// TIA Portal V17 export
// export: Created 2025-03-07T09:17:10.7987229Z, ExportSetting WithDefaults, DisplayName Totally Integrated Automation Portal, DisplayVersion V17 Update 8, DisplayName TIA Portal Openness, DisplayVersion V17 Update 8, DisplayName TIA Portal Version Control Interface, DisplayVersion V17, DisplayName SINAMICS Startdrive Advanced, DisplayVersion V17 SP2, DisplayName SINAMICS Startdrive G110M, G120, G120C, G120D, G120P, G115D, DisplayVersion V17 SP2, DisplayName SINAMICS Startdrive G130, G150, S120, S150, SINAMICS MV, S210, DisplayVersion V17 SP2, DisplayName STEP 7 Professional, DisplayVersion V17 Update 8, DisplayName SINUMERIK ONE STEP 7 Toolbox, DisplayVersion V17 Update 12, DisplayName SINUMERIK 840D sl STEP 7 Toolbox, DisplayVersion V17 Update 12, DisplayName STEP 7 Safety, DisplayVersion V17 Update 6, DisplayName WinCC Advanced, DisplayVersion V17 Update 8
FUNCTION "FC321_CHANNEL_1" : Void   // FC321, LAD
{ S7_Optimized_Access := 'FALSE' }
AUTHOR : ETXETAR
VERSION : 1.0
// stored: AutoNumber false, IsIECCheckEnabled false, SetENOAutomatically false, UDAEnableTagReadback false
BEGIN

REGION Network 1: RESET CHANNEL 1 / CHANNEL 1 (NC RESET - NC START)
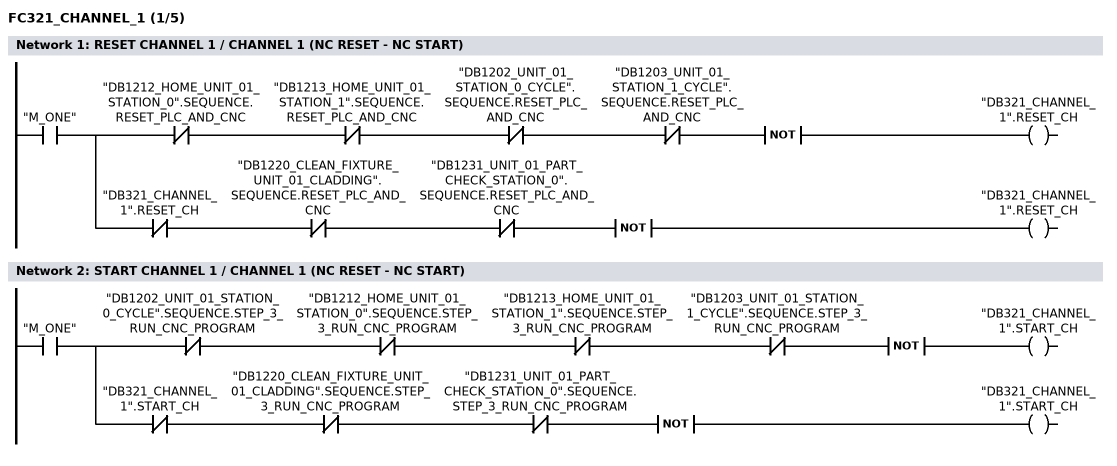
   RUNG wire#powerrail
      Contact( "M_ONE" )
      wire#w1
      I_Contact( "DB1212_HOME_UNIT_01_STATION_0".SEQUENCE.RESET_PLC_AND_CNC )
      I_Contact( "DB1213_HOME_UNIT_01_STATION_1".SEQUENCE.RESET_PLC_AND_CNC )
      I_Contact( "DB1202_UNIT_01_STATION_0_CYCLE".SEQUENCE.RESET_PLC_AND_CNC )
      I_Contact( "DB1203_UNIT_01_STATION_1_CYCLE".SEQUENCE.RESET_PLC_AND_CNC )
      Not()
      Coil( "DB321_CHANNEL_1".RESET_CH )
   END_RUNG
   RUNG wire#w1
      I_Contact( "DB321_CHANNEL_1".RESET_CH )
      I_Contact( "DB1220_CLEAN_FIXTURE_UNIT_01_CLADDING".SEQUENCE.RESET_PLC_AND_CNC )
      I_Contact( "DB1231_UNIT_01_PART_CHECK_STATION_0".SEQUENCE.RESET_PLC_AND_CNC )
      Not()
      Coil( "DB321_CHANNEL_1".RESET_CH )
   END_RUNG
   // the same network as SCL:
   "DB321_CHANNEL_1".RESET_CH := NOT ("M_ONE" AND NOT "DB1212_HOME_UNIT_01_STATION_0".SEQUENCE.RESET_PLC_AND_CNC AND NOT "DB1213_HOME_UNIT_01_STATION_1".SEQUENCE.RESET_PLC_AND_CNC AND NOT "DB1202_UNIT_01_STATION_0_CYCLE".SEQUENCE.RESET_PLC_AND_CNC AND NOT "DB1203_UNIT_01_STATION_1_CYCLE".SEQUENCE.RESET_PLC_AND_CNC);
   "DB321_CHANNEL_1".RESET_CH := NOT ("M_ONE" AND NOT "DB321_CHANNEL_1".RESET_CH AND NOT "DB1220_CLEAN_FIXTURE_UNIT_01_CLADDING".SEQUENCE.RESET_PLC_AND_CNC AND NOT "DB1231_UNIT_01_PART_CHECK_STATION_0".SEQUENCE.RESET_PLC_AND_CNC);
END_REGION

REGION Network 2: START CHANNEL 1 / CHANNEL 1 (NC RESET - NC START)
   RUNG wire#powerrail
      Contact( "M_ONE" )
      wire#w1
      I_Contact( "DB1202_UNIT_01_STATION_0_CYCLE".SEQUENCE.STEP_3_RUN_CNC_PROGRAM )
      I_Contact( "DB1212_HOME_UNIT_01_STATION_0".SEQUENCE.STEP_3_RUN_CNC_PROGRAM )
      I_Contact( "DB1213_HOME_UNIT_01_STATION_1".SEQUENCE.STEP_3_RUN_CNC_PROGRAM )
      I_Contact( "DB1203_UNIT_01_STATION_1_CYCLE".SEQUENCE.STEP_3_RUN_CNC_PROGRAM )
      Not()
      Coil( "DB321_CHANNEL_1".START_CH )
   END_RUNG
   RUNG wire#w1
      I_Contact( "DB321_CHANNEL_1".START_CH )
      I_Contact( "DB1220_CLEAN_FIXTURE_UNIT_01_CLADDING".SEQUENCE.STEP_3_RUN_CNC_PROGRAM )
      I_Contact( "DB1231_UNIT_01_PART_CHECK_STATION_0".SEQUENCE.STEP_3_RUN_CNC_PROGRAM )
      Not()
      Coil( "DB321_CHANNEL_1".START_CH )
   END_RUNG
   // the same network as SCL:
   "DB321_CHANNEL_1".START_CH := NOT ("M_ONE" AND NOT "DB1202_UNIT_01_STATION_0_CYCLE".SEQUENCE.STEP_3_RUN_CNC_PROGRAM AND NOT "DB1212_HOME_UNIT_01_STATION_0".SEQUENCE.STEP_3_RUN_CNC_PROGRAM AND NOT "DB1213_HOME_UNIT_01_STATION_1".SEQUENCE.STEP_3_RUN_CNC_PROGRAM AND NOT "DB1203_UNIT_01_STATION_1_CYCLE".SEQUENCE.STEP_3_RUN_CNC_PROGRAM);
   "DB321_CHANNEL_1".START_CH := NOT ("M_ONE" AND NOT "DB321_CHANNEL_1".START_CH AND NOT "DB1220_CLEAN_FIXTURE_UNIT_01_CLADDING".SEQUENCE.STEP_3_RUN_CNC_PROGRAM AND NOT "DB1231_UNIT_01_PART_CHECK_STATION_0".SEQUENCE.STEP_3_RUN_CNC_PROGRAM);
END_REGION

REGION Network 3: CALL FB321 CHANNEL 1
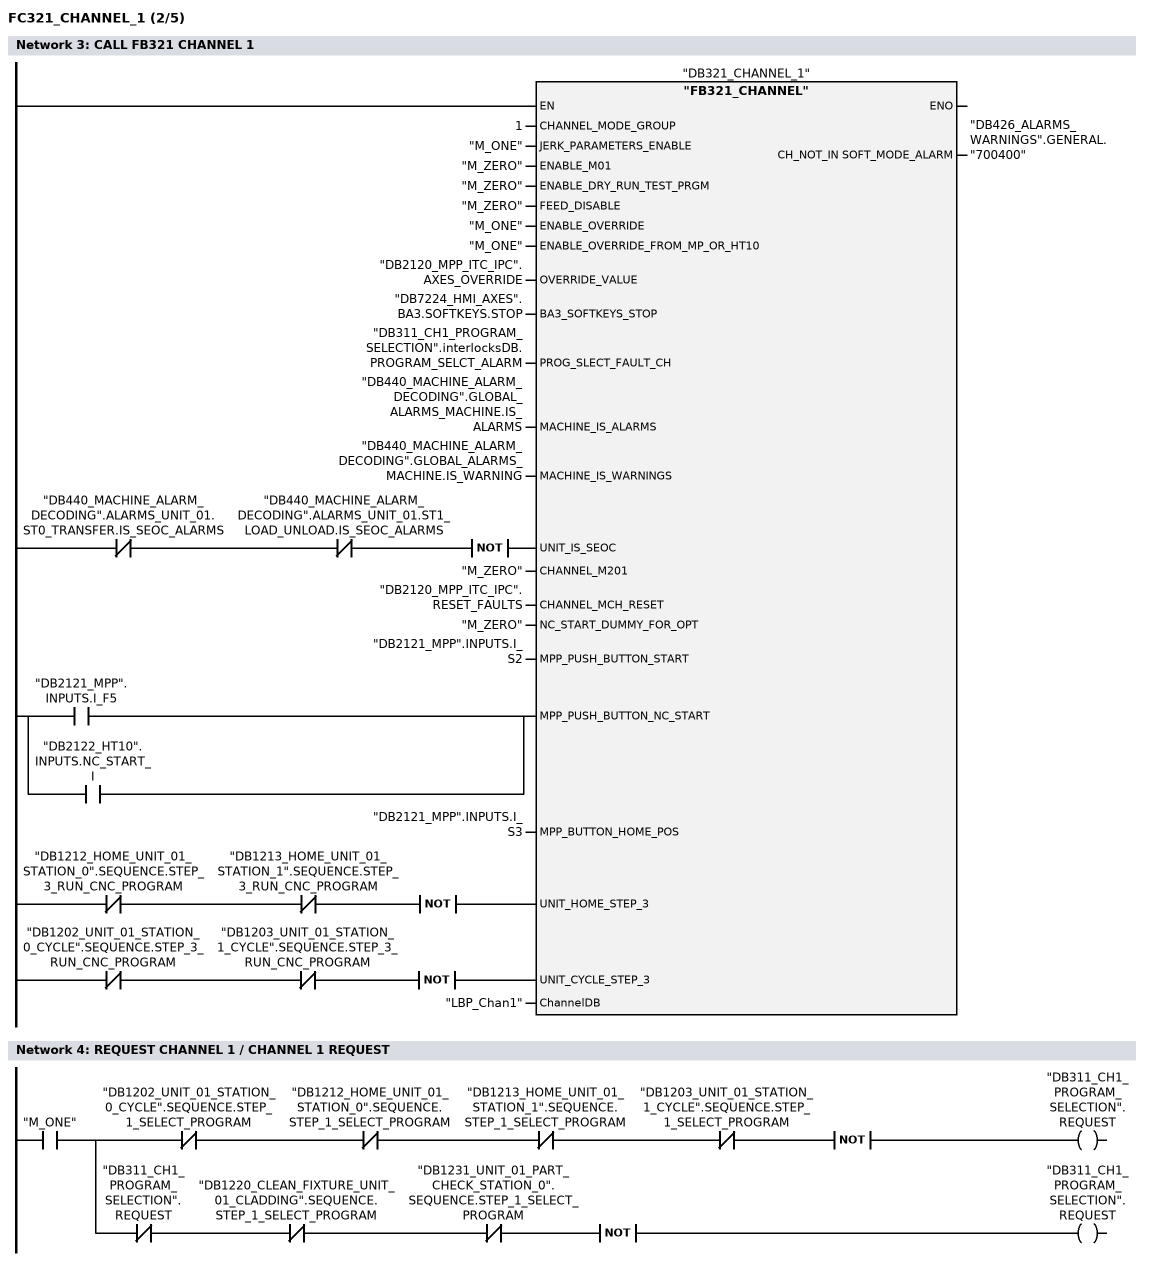
   RUNG wire#powerrail
      "DB321_CHANNEL_1"(UNIT_IS_SEOC := wire#w1, MPP_PUSH_BUTTON_NC_START := wire#w2, UNIT_HOME_STEP_3 := wire#w3, UNIT_CYCLE_STEP_3 := wire#w4, CHANNEL_MODE_GROUP := 1, JERK_PARAMETERS_ENABLE := "M_ONE", ENABLE_M01 := "M_ZERO", ENABLE_DRY_RUN_TEST_PRGM := "M_ZERO", FEED_DISABLE := "M_ZERO", ENABLE_OVERRIDE := "M_ONE", ENABLE_OVERRIDE_FROM_MP_OR_HT10 := "M_ONE", OVERRIDE_VALUE := "DB2120_MPP_ITC_IPC".AXES_OVERRIDE, BA3_SOFTKEYS_STOP := "DB7224_HMI_AXES".BA3.SOFTKEYS.STOP, PROG_SLECT_FAULT_CH := "DB311_CH1_PROGRAM_SELECTION".interlocksDB.PROGRAM_SELCT_ALARM, MACHINE_IS_ALARMS := "DB440_MACHINE_ALARM_DECODING".GLOBAL_ALARMS_MACHINE.IS_ALARMS, MACHINE_IS_WARNINGS := "DB440_MACHINE_ALARM_DECODING".GLOBAL_ALARMS_MACHINE.IS_WARNING, CHANNEL_M201 := "M_ZERO", CHANNEL_MCH_RESET := "DB2120_MPP_ITC_IPC".RESET_FAULTS, NC_START_DUMMY_FOR_OPT := "M_ZERO", MPP_PUSH_BUTTON_START := "DB2121_MPP".INPUTS.I_S2, MPP_BUTTON_HOME_POS := "DB2121_MPP".INPUTS.I_S3, ChannelDB := "LBP_Chan1", "CH_NOT_IN SOFT_MODE_ALARM" => "DB426_ALARMS_WARNINGS".GENERAL."700400")
   END_RUNG
   RUNG wire#powerrail
      I_Contact( "DB440_MACHINE_ALARM_DECODING".ALARMS_UNIT_01.ST0_TRANSFER.IS_SEOC_ALARMS )
      I_Contact( "DB440_MACHINE_ALARM_DECODING".ALARMS_UNIT_01.ST1_LOAD_UNLOAD.IS_SEOC_ALARMS )
      Not()
   END_RUNG wire#w1
   RUNG wire#powerrail
      Contact( "DB2121_MPP".INPUTS.I_F5 )
   END_RUNG wire#w2
   RUNG wire#powerrail
      Contact( "DB2122_HT10".INPUTS.NC_START_I )
   END_RUNG wire#w2
   RUNG wire#powerrail
      I_Contact( "DB1212_HOME_UNIT_01_STATION_0".SEQUENCE.STEP_3_RUN_CNC_PROGRAM )
      I_Contact( "DB1213_HOME_UNIT_01_STATION_1".SEQUENCE.STEP_3_RUN_CNC_PROGRAM )
      Not()
   END_RUNG wire#w3
   RUNG wire#powerrail
      I_Contact( "DB1202_UNIT_01_STATION_0_CYCLE".SEQUENCE.STEP_3_RUN_CNC_PROGRAM )
      I_Contact( "DB1203_UNIT_01_STATION_1_CYCLE".SEQUENCE.STEP_3_RUN_CNC_PROGRAM )
      Not()
   END_RUNG wire#w4
   // the same network as SCL:
   "DB321_CHANNEL_1"(CHANNEL_MODE_GROUP := 1,   // "FB321_CHANNEL"
                     JERK_PARAMETERS_ENABLE := "M_ONE",
                     ENABLE_M01 := "M_ZERO",
                     ENABLE_DRY_RUN_TEST_PRGM := "M_ZERO",
                     FEED_DISABLE := "M_ZERO",
                     ENABLE_OVERRIDE := "M_ONE",
                     ENABLE_OVERRIDE_FROM_MP_OR_HT10 := "M_ONE",
                     OVERRIDE_VALUE := "DB2120_MPP_ITC_IPC".AXES_OVERRIDE,
                     BA3_SOFTKEYS_STOP := "DB7224_HMI_AXES".BA3.SOFTKEYS.STOP,
                     PROG_SLECT_FAULT_CH := "DB311_CH1_PROGRAM_SELECTION".interlocksDB.PROGRAM_SELCT_ALARM,
                     MACHINE_IS_ALARMS := "DB440_MACHINE_ALARM_DECODING".GLOBAL_ALARMS_MACHINE.IS_ALARMS,
                     MACHINE_IS_WARNINGS := "DB440_MACHINE_ALARM_DECODING".GLOBAL_ALARMS_MACHINE.IS_WARNING,
                     UNIT_IS_SEOC := NOT (NOT "DB440_MACHINE_ALARM_DECODING".ALARMS_UNIT_01.ST0_TRANSFER.IS_SEOC_ALARMS AND NOT "DB440_MACHINE_ALARM_DECODING".ALARMS_UNIT_01.ST1_LOAD_UNLOAD.IS_SEOC_ALARMS),
                     CHANNEL_M201 := "M_ZERO",
                     CHANNEL_MCH_RESET := "DB2120_MPP_ITC_IPC".RESET_FAULTS,
                     NC_START_DUMMY_FOR_OPT := "M_ZERO",
                     MPP_PUSH_BUTTON_START := "DB2121_MPP".INPUTS.I_S2,
                     MPP_PUSH_BUTTON_NC_START := "DB2121_MPP".INPUTS.I_F5 OR "DB2122_HT10".INPUTS.NC_START_I,
                     MPP_BUTTON_HOME_POS := "DB2121_MPP".INPUTS.I_S3,
                     UNIT_HOME_STEP_3 := NOT (NOT "DB1212_HOME_UNIT_01_STATION_0".SEQUENCE.STEP_3_RUN_CNC_PROGRAM AND NOT "DB1213_HOME_UNIT_01_STATION_1".SEQUENCE.STEP_3_RUN_CNC_PROGRAM),
                     UNIT_CYCLE_STEP_3 := NOT (NOT "DB1202_UNIT_01_STATION_0_CYCLE".SEQUENCE.STEP_3_RUN_CNC_PROGRAM AND NOT "DB1203_UNIT_01_STATION_1_CYCLE".SEQUENCE.STEP_3_RUN_CNC_PROGRAM),
                     ChannelDB := "LBP_Chan1",
                     "CH_NOT_IN SOFT_MODE_ALARM" => "DB426_ALARMS_WARNINGS".GENERAL."700400");
END_REGION

REGION Network 4: REQUEST CHANNEL 1 / CHANNEL 1 REQUEST
   RUNG wire#powerrail
      Contact( "M_ONE" )
      wire#w1
      I_Contact( "DB1202_UNIT_01_STATION_0_CYCLE".SEQUENCE.STEP_1_SELECT_PROGRAM )
      I_Contact( "DB1212_HOME_UNIT_01_STATION_0".SEQUENCE.STEP_1_SELECT_PROGRAM )
      I_Contact( "DB1213_HOME_UNIT_01_STATION_1".SEQUENCE.STEP_1_SELECT_PROGRAM )
      I_Contact( "DB1203_UNIT_01_STATION_1_CYCLE".SEQUENCE.STEP_1_SELECT_PROGRAM )
      Not()
      Coil( "DB311_CH1_PROGRAM_SELECTION".REQUEST )
   END_RUNG
   RUNG wire#w1
      I_Contact( "DB311_CH1_PROGRAM_SELECTION".REQUEST )
      I_Contact( "DB1220_CLEAN_FIXTURE_UNIT_01_CLADDING".SEQUENCE.STEP_1_SELECT_PROGRAM )
      I_Contact( "DB1231_UNIT_01_PART_CHECK_STATION_0".SEQUENCE.STEP_1_SELECT_PROGRAM )
      Not()
      Coil( "DB311_CH1_PROGRAM_SELECTION".REQUEST )
   END_RUNG
   // the same network as SCL:
   "DB311_CH1_PROGRAM_SELECTION".REQUEST := NOT ("M_ONE" AND NOT "DB1202_UNIT_01_STATION_0_CYCLE".SEQUENCE.STEP_1_SELECT_PROGRAM AND NOT "DB1212_HOME_UNIT_01_STATION_0".SEQUENCE.STEP_1_SELECT_PROGRAM AND NOT "DB1213_HOME_UNIT_01_STATION_1".SEQUENCE.STEP_1_SELECT_PROGRAM AND NOT "DB1203_UNIT_01_STATION_1_CYCLE".SEQUENCE.STEP_1_SELECT_PROGRAM);
   "DB311_CH1_PROGRAM_SELECTION".REQUEST := NOT ("M_ONE" AND NOT "DB311_CH1_PROGRAM_SELECTION".REQUEST AND NOT "DB1220_CLEAN_FIXTURE_UNIT_01_CLADDING".SEQUENCE.STEP_1_SELECT_PROGRAM AND NOT "DB1231_UNIT_01_PART_CHECK_STATION_0".SEQUENCE.STEP_1_SELECT_PROGRAM);
END_REGION

REGION Network 5: CALL FB311 CHANNEL PROGRAM SELECTION / CHANNEL 1
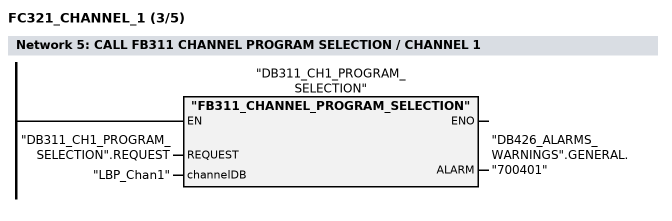
   RUNG wire#powerrail
      "DB311_CH1_PROGRAM_SELECTION"(REQUEST := "DB311_CH1_PROGRAM_SELECTION".REQUEST, channelDB := "LBP_Chan1", ALARM => "DB426_ALARMS_WARNINGS".GENERAL."700401")
   END_RUNG
   // the same network as SCL:
   "DB311_CH1_PROGRAM_SELECTION"(REQUEST := "DB311_CH1_PROGRAM_SELECTION".REQUEST,   // "FB311_CHANNEL_PROGRAM_SELECTION"
                           channelDB := "LBP_Chan1",
                           ALARM => "DB426_ALARMS_WARNINGS".GENERAL."700401");
END_REGION

REGION Network 6: CALL FB301 CHANNEL READ AXES POSITIONS
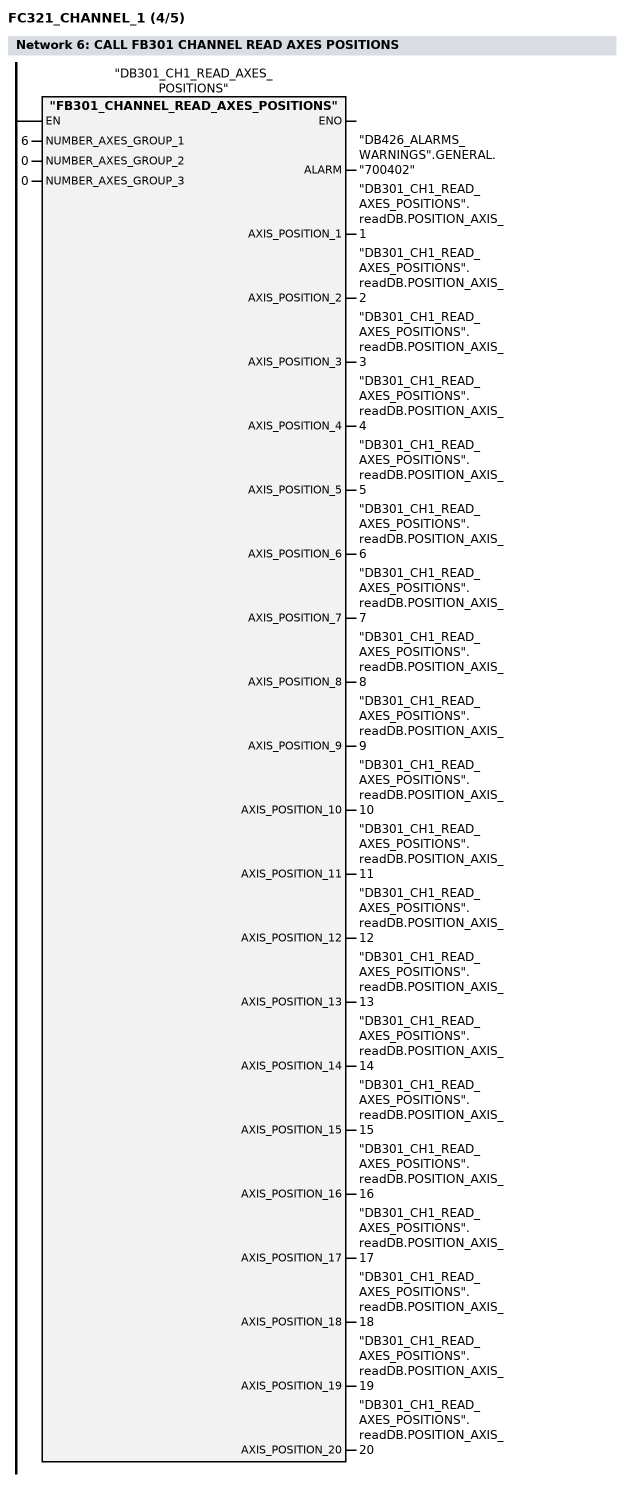
   RUNG wire#powerrail
      "DB301_CH1_READ_AXES_POSITIONS"(NUMBER_AXES_GROUP_1 := 6, NUMBER_AXES_GROUP_2 := 0, NUMBER_AXES_GROUP_3 := 0, ALARM => "DB426_ALARMS_WARNINGS".GENERAL."700402", AXIS_POSITION_1 => "DB301_CH1_READ_AXES_POSITIONS".readDB.POSITION_AXIS_1, AXIS_POSITION_2 => "DB301_CH1_READ_AXES_POSITIONS".readDB.POSITION_AXIS_2, AXIS_POSITION_3 => "DB301_CH1_READ_AXES_POSITIONS".readDB.POSITION_AXIS_3, AXIS_POSITION_4 => "DB301_CH1_READ_AXES_POSITIONS".readDB.POSITION_AXIS_4, AXIS_POSITION_5 => "DB301_CH1_READ_AXES_POSITIONS".readDB.POSITION_AXIS_5, AXIS_POSITION_6 => "DB301_CH1_READ_AXES_POSITIONS".readDB.POSITION_AXIS_6, AXIS_POSITION_7 => "DB301_CH1_READ_AXES_POSITIONS".readDB.POSITION_AXIS_7, AXIS_POSITION_8 => "DB301_CH1_READ_AXES_POSITIONS".readDB.POSITION_AXIS_8, AXIS_POSITION_9 => "DB301_CH1_READ_AXES_POSITIONS".readDB.POSITION_AXIS_9, AXIS_POSITION_10 => "DB301_CH1_READ_AXES_POSITIONS".readDB.POSITION_AXIS_10, AXIS_POSITION_11 => "DB301_CH1_READ_AXES_POSITIONS".readDB.POSITION_AXIS_11, AXIS_POSITION_12 => "DB301_CH1_READ_AXES_POSITIONS".readDB.POSITION_AXIS_12, AXIS_POSITION_13 => "DB301_CH1_READ_AXES_POSITIONS".readDB.POSITION_AXIS_13, AXIS_POSITION_14 => "DB301_CH1_READ_AXES_POSITIONS".readDB.POSITION_AXIS_14, AXIS_POSITION_15 => "DB301_CH1_READ_AXES_POSITIONS".readDB.POSITION_AXIS_15, AXIS_POSITION_16 => "DB301_CH1_READ_AXES_POSITIONS".readDB.POSITION_AXIS_16, AXIS_POSITION_17 => "DB301_CH1_READ_AXES_POSITIONS".readDB.POSITION_AXIS_17, AXIS_POSITION_18 => "DB301_CH1_READ_AXES_POSITIONS".readDB.POSITION_AXIS_18, AXIS_POSITION_19 => "DB301_CH1_READ_AXES_POSITIONS".readDB.POSITION_AXIS_19, AXIS_POSITION_20 => "DB301_CH1_READ_AXES_POSITIONS".readDB.POSITION_AXIS_20)
   END_RUNG
   // the same network as SCL:
   "DB301_CH1_READ_AXES_POSITIONS"(NUMBER_AXES_GROUP_1 := 6,   // "FB301_CHANNEL_READ_AXES_POSITIONS"
                           NUMBER_AXES_GROUP_2 := 0,
                           NUMBER_AXES_GROUP_3 := 0,
                           ALARM => "DB426_ALARMS_WARNINGS".GENERAL."700402",
                           AXIS_POSITION_1 => "DB301_CH1_READ_AXES_POSITIONS".readDB.POSITION_AXIS_1,
                           AXIS_POSITION_2 => "DB301_CH1_READ_AXES_POSITIONS".readDB.POSITION_AXIS_2,
                           AXIS_POSITION_3 => "DB301_CH1_READ_AXES_POSITIONS".readDB.POSITION_AXIS_3,
                           AXIS_POSITION_4 => "DB301_CH1_READ_AXES_POSITIONS".readDB.POSITION_AXIS_4,
                           AXIS_POSITION_5 => "DB301_CH1_READ_AXES_POSITIONS".readDB.POSITION_AXIS_5,
                           AXIS_POSITION_6 => "DB301_CH1_READ_AXES_POSITIONS".readDB.POSITION_AXIS_6,
                           AXIS_POSITION_7 => "DB301_CH1_READ_AXES_POSITIONS".readDB.POSITION_AXIS_7,
                           AXIS_POSITION_8 => "DB301_CH1_READ_AXES_POSITIONS".readDB.POSITION_AXIS_8,
                           AXIS_POSITION_9 => "DB301_CH1_READ_AXES_POSITIONS".readDB.POSITION_AXIS_9,
                           AXIS_POSITION_10 => "DB301_CH1_READ_AXES_POSITIONS".readDB.POSITION_AXIS_10,
                           AXIS_POSITION_11 => "DB301_CH1_READ_AXES_POSITIONS".readDB.POSITION_AXIS_11,
                           AXIS_POSITION_12 => "DB301_CH1_READ_AXES_POSITIONS".readDB.POSITION_AXIS_12,
                           AXIS_POSITION_13 => "DB301_CH1_READ_AXES_POSITIONS".readDB.POSITION_AXIS_13,
                           AXIS_POSITION_14 => "DB301_CH1_READ_AXES_POSITIONS".readDB.POSITION_AXIS_14,
                           AXIS_POSITION_15 => "DB301_CH1_READ_AXES_POSITIONS".readDB.POSITION_AXIS_15,
                           AXIS_POSITION_16 => "DB301_CH1_READ_AXES_POSITIONS".readDB.POSITION_AXIS_16,
                           AXIS_POSITION_17 => "DB301_CH1_READ_AXES_POSITIONS".readDB.POSITION_AXIS_17,
                           AXIS_POSITION_18 => "DB301_CH1_READ_AXES_POSITIONS".readDB.POSITION_AXIS_18,
                           AXIS_POSITION_19 => "DB301_CH1_READ_AXES_POSITIONS".readDB.POSITION_AXIS_19,
                           AXIS_POSITION_20 => "DB301_CH1_READ_AXES_POSITIONS".readDB.POSITION_AXIS_20);
END_REGION

REGION Network 7: CALL FC341 NCK M STA 0 / CALL FC1181
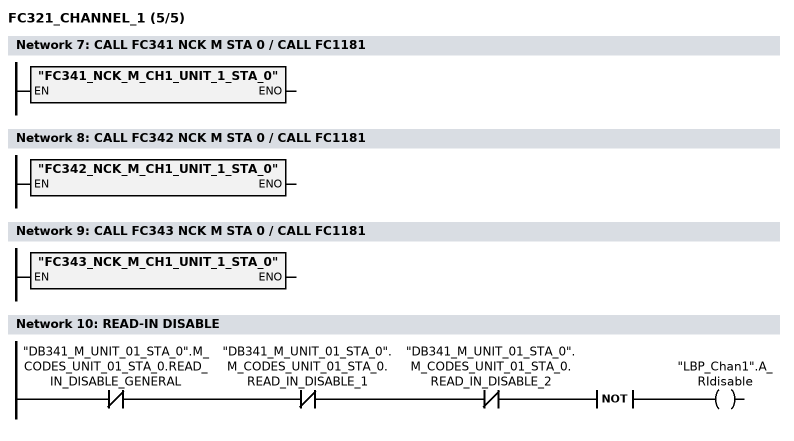
   RUNG wire#powerrail
      "FC341_NCK_M_CH1_UNIT_1_STA_0"()
   END_RUNG
   // the same network as SCL:
   "FC341_NCK_M_CH1_UNIT_1_STA_0"();
END_REGION

REGION Network 8: CALL FC342 NCK M STA 0 / CALL FC1181
   RUNG wire#powerrail
      "FC342_NCK_M_CH1_UNIT_1_STA_0"()
   END_RUNG
   // the same network as SCL:
   "FC342_NCK_M_CH1_UNIT_1_STA_0"();
END_REGION

REGION Network 9: CALL FC343 NCK M STA 0 / CALL FC1181
   RUNG wire#powerrail
      "FC343_NCK_M_CH1_UNIT_1_STA_0"()
   END_RUNG
   // the same network as SCL:
   "FC343_NCK_M_CH1_UNIT_1_STA_0"();
END_REGION

REGION Network 10: READ-IN DISABLE
   RUNG wire#powerrail
      I_Contact( "DB341_M_UNIT_01_STA_0".M_CODES_UNIT_01_STA_0.READ_IN_DISABLE_GENERAL )
      I_Contact( "DB341_M_UNIT_01_STA_0".M_CODES_UNIT_01_STA_0.READ_IN_DISABLE_1 )
      I_Contact( "DB341_M_UNIT_01_STA_0".M_CODES_UNIT_01_STA_0.READ_IN_DISABLE_2 )
      Not()
      Coil( "LBP_Chan1".A_RIdisable )
   END_RUNG
   // the same network as SCL:
   "LBP_Chan1".A_RIdisable := NOT (NOT "DB341_M_UNIT_01_STA_0".M_CODES_UNIT_01_STA_0.READ_IN_DISABLE_GENERAL AND NOT "DB341_M_UNIT_01_STA_0".M_CODES_UNIT_01_STA_0.READ_IN_DISABLE_1 AND NOT "DB341_M_UNIT_01_STA_0".M_CODES_UNIT_01_STA_0.READ_IN_DISABLE_2);
END_REGION
END_FUNCTION
